FUNCTION maximum : DINT
VAR_INPUT
END_VAR
VAR
	temp : DINT;
END_VAR

temp := MAX(Glbl.state1Counter, Glbl.state2Counter);
temp := MAX(Glbl.state3Counter, temp);
temp := MAX(Glbl.state4Counter, temp);
temp := MAX(Glbl.state5Counter, temp);
temp := MAX(Glbl.state6Counter, temp);
temp := MAX(Glbl.state7Counter, temp);
temp := MAX(Glbl.state8Counter, temp);
maximum := temp;

END_FUNCTION

(* stored: Version 1.1.0.1, ProductVersion 3.1.4022.10
   POU maximum: Id {59ca9b71-0d0a-41a3-9b92-9bb620fb7ead}, SpecialFunc None *)
